// TIA Portal project "zamanlayıcılar" (V16)

(* hardware
DEVICE "S71500/ET200MP station_1"  S7-1500 station
   slot 0: "Rail_0"  Rack  6ES7 590-1***0-0AA0
   slot 1: "PLC_1"  CPU 1511C-1 PN  6ES7 511-1CK00-0AB0  V2.8
      slot 3: "CPU display_1"  6ES7591-1AA00-0AA0
      slot 32768: "PROFINET interface_1"  X1
         slot 32769: "Port_1"  X1 P1
         slot 32770: "Port_2"  X1 P2
      slot 34817: "Virtual CP interface port_1"  Virtual CP interface port  Virtual CP interface port
*)

// ===== PLC "PLC_1"  CPU 1511C-1 PN =====

VAR_GLOBAL   // PLC tag table "Default tag table"
   "start" AT %I0.0 : Bool;
   "motor1" AT %Q0.1 : Bool;
   "motor2" AT %Q0.2 : Bool;
   "motor3" AT %Q0.3 : Bool;
   "yr1" AT %M0.0 : Bool;
   "stop" AT %I0.1 : Bool;
END_VAR

// folder: System blocks/Program resources

DATA_BLOCK "dzr1"   // DB1
{ S7_Optimized_Access := 'TRUE' }
AUTHOR : Simatic
FAMILY : IEC
NAME : IEC_TMR
VERSION : 1.0
// stored: InstanceOfName IEC_TIMER
"IEC_TIMER"
BEGIN
END_DATA_BLOCK

DATA_BLOCK "dzr2"   // DB2
{ S7_Optimized_Access := 'TRUE' }
AUTHOR : Simatic
FAMILY : IEC
NAME : IEC_TMR
VERSION : 1.0
// stored: InstanceOfName IEC_TIMER
"IEC_TIMER"
BEGIN
END_DATA_BLOCK

DATA_BLOCK "tzr1"   // DB3
{ S7_Optimized_Access := 'TRUE' }
AUTHOR : Simatic
FAMILY : IEC
NAME : IEC_TMR
VERSION : 1.0
// stored: InstanceOfName IEC_TIMER
"IEC_TIMER"
BEGIN
END_DATA_BLOCK

DATA_BLOCK "dzr3"   // DB4
{ S7_Optimized_Access := 'TRUE' }
AUTHOR : Simatic
FAMILY : IEC
NAME : IEC_TMR
VERSION : 1.0
// stored: InstanceOfName IEC_TIMER
"IEC_TIMER"
BEGIN
END_DATA_BLOCK

// folder: (top level)

ORGANIZATION_BLOCK "Main"   // OB1, LAD, ProgramCycle
TITLE = "Main Program Sweep (Cycle)"
{ S7_Optimized_Access := 'TRUE' }
VERSION : 0.1
   VAR_INPUT
      Initial_Call : Bool;   // Initial call of this OB
      Remanence : Bool;   // =True, if remanent data are available
   END_VAR
BEGIN

REGION Network 1
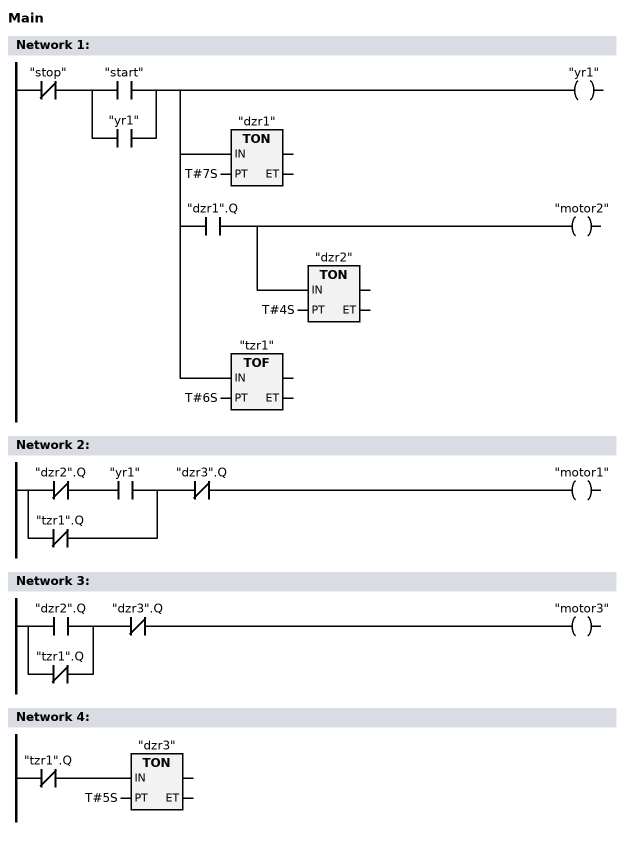
   "yr1" := NOT "stop" AND ("start" OR "yr1");
   "dzr1".TON(IN := "yr1", PT := T#7S);
   "motor2" := "yr1" AND "dzr1".Q;
   "dzr2".TON(IN := "motor2", PT := T#4S);
   "tzr1".TOF(IN := "yr1", PT := T#6S);
END_REGION

REGION Network 2
   RUNG wire#powerrail
      I_Contact( "dzr2".Q )
      Contact( "yr1" )
      wire#w1
      I_Contact( "dzr3".Q )
      Coil( "motor1" )
   END_RUNG
   RUNG wire#powerrail
      I_Contact( "tzr1".Q )
   END_RUNG wire#w1
   // the same network as SCL:
   "motor1" := ((NOT "dzr2".Q AND "yr1") OR NOT "tzr1".Q) AND NOT "dzr3".Q;
END_REGION

REGION Network 3
   RUNG wire#powerrail
      Contact( "dzr2".Q )
      wire#w1
      I_Contact( "dzr3".Q )
      Coil( "motor3" )
   END_RUNG
   RUNG wire#powerrail
      I_Contact( "tzr1".Q )
   END_RUNG wire#w1
   // the same network as SCL:
   "motor3" := ("dzr2".Q OR NOT "tzr1".Q) AND NOT "dzr3".Q;
END_REGION

REGION Network 4
   "dzr3".TON(IN := NOT "tzr1".Q, PT := T#5S);
END_REGION
END_ORGANIZATION_BLOCK